FUNCTION INTERNAL _RegSignal : Result
VAR_INPUT
    iSignal : I_SignalNode;
END_VAR
VAR_OUTPUT
	nIndex	: UDINT;
END_VAR

IF NOT _Runtime.bInit THEN
	_RegSignal := Err.Init;
	RETURN;
END_IF

IF iSignal = 0 THEN
	_RegSignal := Err.Itf0;
	RETURN;
END_IF

IF _Broadcast.nSignalLen = Param.SIGNAL_CAP THEN
	_RegSignal := Err.Ovf;
	RETURN;
END_IF

_Broadcast.nSignalLen := _Broadcast.nSignalLen + 1;
_Broadcast.iSignal[_Broadcast.nSignalLen] := iSignal;
nIndex := _Broadcast.nSignalLen;
_RegSignal := Ok;

END_FUNCTION

(* stored: Version 1.1.0.1
   POU _RegSignal: Id {cde70202-4e07-4c54-9336-33c9199281ce}, SpecialFunc None *)
